(* PLC project Unnamed, Unknown Unnamed 1 *)
(* stored: creationDateTime 2023-03-10T10:37:17, modificationDateTime 2023-03-15T15:56:42 *)

(* SIEMENS AG- Beispielprogramm *)
FUNCTION_BLOCK Roll_Down_Shutters
  VAR_INPUT
    IN1 : BOOL;
    IN2 : BOOL;
    IN3 : BOOL;
    IN4 : BOOL;
    IN5 : BOOL;
    IN6 : BOOL;
    TIME14 : BOOL;
    TIME4 : BOOL;
  END_VAR
  VAR_OUTPUT
    OUT1 : BOOL;
    OUT2 : BOOL;
  END_VAR
  VAR  (* added by the conversion: wires and edge detectors of the diagram *)
    _AND35_OUT : BOOL;
  END_VAR

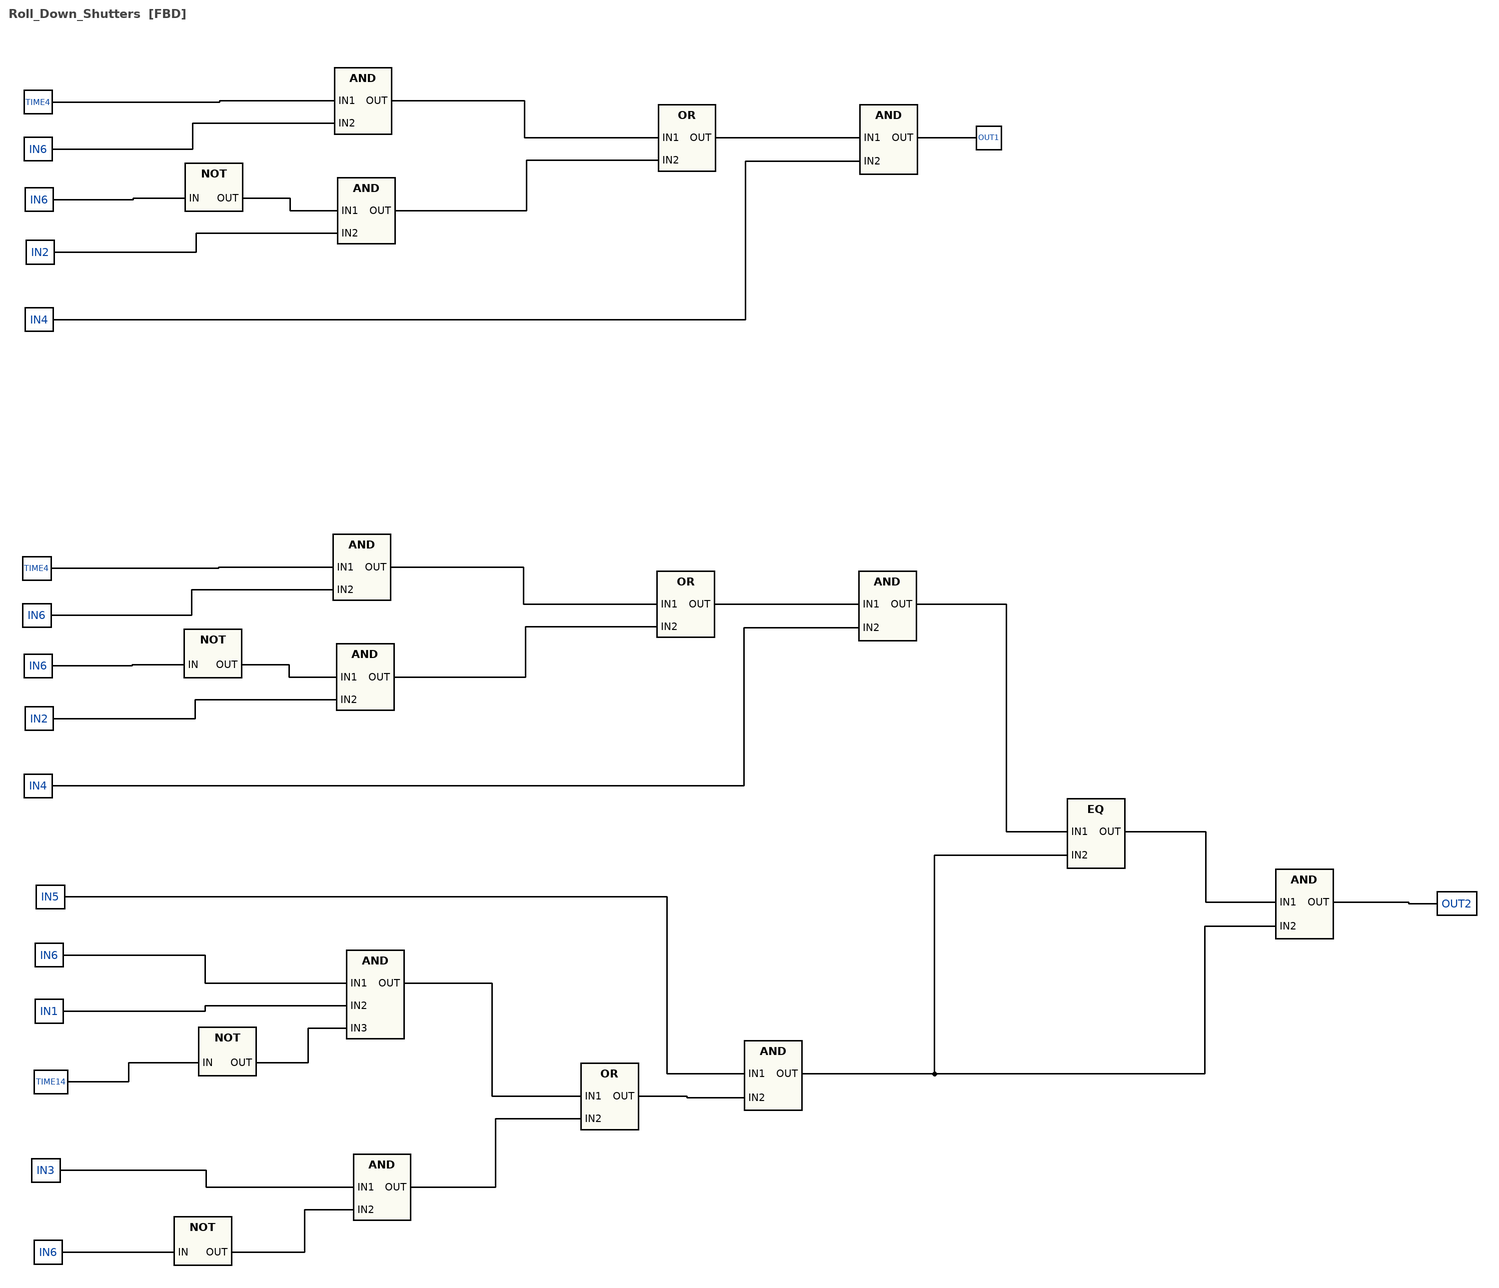
(* FBD diagram, written out as Structured Text *)
OUT1 := (TIME4 AND IN6 OR NOT IN6 AND IN2) AND IN4;
_AND35_OUT := IN5 AND (IN6 AND IN1 AND NOT TIME14 OR IN3 AND NOT IN6);
OUT2 := ((TIME4 AND IN6 OR NOT IN6 AND IN2) AND IN4) = _AND35_OUT AND _AND35_OUT;
END_FUNCTION_BLOCK

CONFIGURATION config
  RESOURCE resource1 ON PLC
  END_RESOURCE
END_CONFIGURATION
